// TIA Portal V19 export
FUNCTION "Mode Selection" : Void   // FC4, LAD
{ S7_Optimized_Access := 'TRUE' }
// stored: SetENOAutomatically false
   VAR_TEMP   // added for the SCL form of the ladder/FBD networks
      _w1 : Bool;
   END_VAR
BEGIN

REGION Network 1: MFG STAND BY
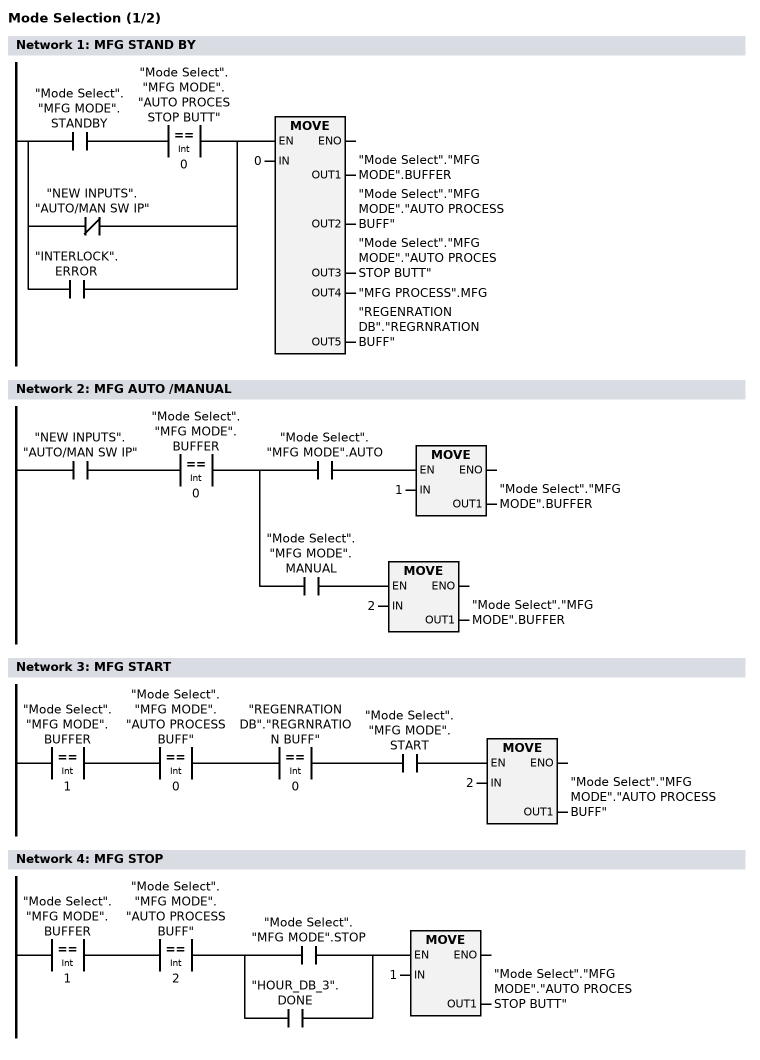
   RUNG wire#powerrail
      Contact( "Mode Select"."MFG MODE".STANDBY )
      { S7_Templates := "SrcType := Int" } EQ_Contact(in1 := "Mode Select"."MFG MODE"."AUTO PROCES STOP BUTT", in2 := 0)
      wire#w1
      Move(in := 0, out1 => "Mode Select"."MFG MODE".BUFFER, out2 => "Mode Select"."MFG MODE"."AUTO PROCESS BUFF", out3 => "Mode Select"."MFG MODE"."AUTO PROCES STOP BUTT", out4 => "MFG PROCESS".MFG, out5 => "REGENRATION DB"."REGRNRATION BUFF")
   END_RUNG
   RUNG wire#powerrail
      I_Contact( "NEW INPUTS"."AUTO/MAN SW IP" )
   END_RUNG wire#w1
   RUNG wire#powerrail
      Contact( "INTERLOCK".ERROR )
   END_RUNG wire#w1
   // the same network as SCL:
   IF ("Mode Select"."MFG MODE".STANDBY AND ("Mode Select"."MFG MODE"."AUTO PROCES STOP BUTT" = 0)) OR NOT "NEW INPUTS"."AUTO/MAN SW IP" OR "INTERLOCK".ERROR THEN
       "Mode Select"."MFG MODE".BUFFER := 0;
       "Mode Select"."MFG MODE"."AUTO PROCESS BUFF" := 0;
       "Mode Select"."MFG MODE"."AUTO PROCES STOP BUTT" := 0;
       "MFG PROCESS".MFG := 0;
       "REGENRATION DB"."REGRNRATION BUFF" := 0;
   END_IF;
END_REGION

REGION Network 2: MFG AUTO /MANUAL
   RUNG wire#powerrail
      Contact( "NEW INPUTS"."AUTO/MAN SW IP" )
      { S7_Templates := "SrcType := Int" } EQ_Contact(in1 := "Mode Select"."MFG MODE".BUFFER, in2 := 0)
      wire#w1
      Contact( "Mode Select"."MFG MODE".AUTO )
      Move(in := 1, out1 => "Mode Select"."MFG MODE".BUFFER)
   END_RUNG
   RUNG wire#w1
      Contact( "Mode Select"."MFG MODE".MANUAL )
      Move(in := 2, out1 => "Mode Select"."MFG MODE".BUFFER)
   END_RUNG
   // the same network as SCL:
   #_w1 := "NEW INPUTS"."AUTO/MAN SW IP" AND ("Mode Select"."MFG MODE".BUFFER = 0);
   IF #_w1 AND "Mode Select"."MFG MODE".AUTO THEN "Mode Select"."MFG MODE".BUFFER := 1; END_IF;
   IF #_w1 AND "Mode Select"."MFG MODE".MANUAL THEN "Mode Select"."MFG MODE".BUFFER := 2; END_IF;
END_REGION

REGION Network 3: MFG START
   RUNG wire#powerrail
      { S7_Templates := "SrcType := Int" } EQ_Contact(in1 := "Mode Select"."MFG MODE".BUFFER, in2 := 1)
      { S7_Templates := "SrcType := Int" } EQ_Contact(in1 := "Mode Select"."MFG MODE"."AUTO PROCESS BUFF", in2 := 0)
      { S7_Templates := "SrcType := Int" } EQ_Contact(in1 := "REGENRATION DB"."REGRNRATION BUFF", in2 := 0)
      Contact( "Mode Select"."MFG MODE".START )
      Move(in := 2, out1 => "Mode Select"."MFG MODE"."AUTO PROCESS BUFF")
   END_RUNG
   // the same network as SCL:
   IF ("Mode Select"."MFG MODE".BUFFER = 1) AND ("Mode Select"."MFG MODE"."AUTO PROCESS BUFF" = 0) AND ("REGENRATION DB"."REGRNRATION BUFF" = 0) AND "Mode Select"."MFG MODE".START THEN
       "Mode Select"."MFG MODE"."AUTO PROCESS BUFF" := 2;
   END_IF;
END_REGION

REGION Network 4: MFG STOP
   RUNG wire#powerrail
      { S7_Templates := "SrcType := Int" } EQ_Contact(in1 := "Mode Select"."MFG MODE".BUFFER, in2 := 1)
      { S7_Templates := "SrcType := Int" } EQ_Contact(in1 := "Mode Select"."MFG MODE"."AUTO PROCESS BUFF", in2 := 2)
      wire#w1
      Contact( "Mode Select"."MFG MODE".STOP )
      wire#w2
      Move(in := 1, out1 => "Mode Select"."MFG MODE"."AUTO PROCES STOP BUTT")
   END_RUNG
   RUNG wire#w1
      Contact( "HOUR_DB_3".DONE )
   END_RUNG wire#w2
   // the same network as SCL:
   IF ("Mode Select"."MFG MODE".BUFFER = 1) AND ("Mode Select"."MFG MODE"."AUTO PROCESS BUFF" = 2) AND ("Mode Select"."MFG MODE".STOP OR "HOUR_DB_3".DONE) THEN
       "Mode Select"."MFG MODE"."AUTO PROCES STOP BUTT" := 1;
   END_IF;
END_REGION

REGION Network 5: STOP MGF ALL PROCESS
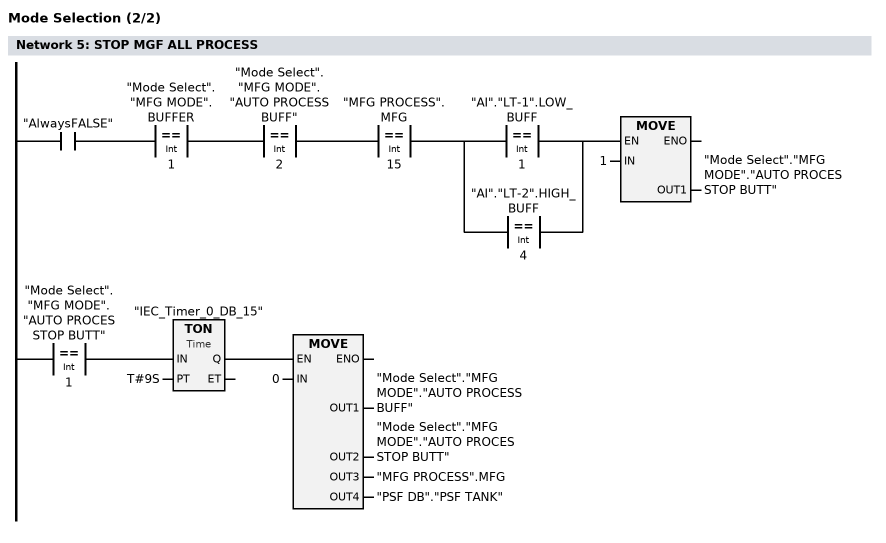
   RUNG wire#powerrail
      Contact( "AlwaysFALSE" )
      { S7_Templates := "SrcType := Int" } EQ_Contact(in1 := "Mode Select"."MFG MODE".BUFFER, in2 := 1)
      { S7_Templates := "SrcType := Int" } EQ_Contact(in1 := "Mode Select"."MFG MODE"."AUTO PROCESS BUFF", in2 := 2)
      { S7_Templates := "SrcType := Int" } EQ_Contact(in1 := "MFG PROCESS".MFG, in2 := 15)
      wire#w1
      { S7_Templates := "SrcType := Int" } EQ_Contact(in1 := "AI"."LT-1".LOW_BUFF, in2 := 1)
      wire#w2
      Move(in := 1, out1 => "Mode Select"."MFG MODE"."AUTO PROCES STOP BUTT")
   END_RUNG
   RUNG wire#w1
      { S7_Templates := "SrcType := Int" } EQ_Contact(in1 := "AI"."LT-2".HIGH_BUFF, in2 := 4)
   END_RUNG wire#w2
   RUNG wire#powerrail
      { S7_Templates := "SrcType := Int" } EQ_Contact(in1 := "Mode Select"."MFG MODE"."AUTO PROCES STOP BUTT", in2 := 1)
      { S7_Templates := "time_type := Time" } "IEC_Timer_0_DB_15".TON(pt := T#9S, et =>)
      Move(in := 0, out1 => "Mode Select"."MFG MODE"."AUTO PROCESS BUFF", out2 => "Mode Select"."MFG MODE"."AUTO PROCES STOP BUTT", out3 => "MFG PROCESS".MFG, out4 => "PSF DB"."PSF TANK")
   END_RUNG
   // the same network as SCL:
   IF "AlwaysFALSE" AND ("Mode Select"."MFG MODE".BUFFER = 1) AND ("Mode Select"."MFG MODE"."AUTO PROCESS BUFF" = 2) AND ("MFG PROCESS".MFG = 15) AND (("AI"."LT-1".LOW_BUFF = 1) OR ("AI"."LT-2".HIGH_BUFF = 4)) THEN
       "Mode Select"."MFG MODE"."AUTO PROCES STOP BUTT" := 1;
   END_IF;
   "IEC_Timer_0_DB_15".TON(IN := "Mode Select"."MFG MODE"."AUTO PROCES STOP BUTT" = 1, PT := T#9S);
   IF "IEC_Timer_0_DB_15".Q THEN
       "Mode Select"."MFG MODE"."AUTO PROCESS BUFF" := 0;
       "Mode Select"."MFG MODE"."AUTO PROCES STOP BUTT" := 0;
       "MFG PROCESS".MFG := 0;
       "PSF DB"."PSF TANK" := 0;
   END_IF;
END_REGION
END_FUNCTION
